// TIA Portal V17 export
// export: Created 2023-02-14T02:49:15.3088685Z, ExportSetting WithDefaults, DisplayName Totally Integrated Automation Portal, DisplayVersion V17, DisplayName TIA Portal Openness, DisplayVersion V17, DisplayName TIA Portal Teamcenter Gateway, DisplayVersion V17, DisplayName TIA Portal Version Control Interface, DisplayVersion V17, DisplayName SINAMICS Startdrive Advanced, DisplayVersion V17, DisplayName SINAMICS Startdrive G130, G150, S120, S150, SINAMICS MV, S210, DisplayVersion V17, DisplayName SINAMICS Startdrive G110M, G120, G120C, G120D, G120P, G115D, DisplayVersion V17, DisplayName STEP 7 Professional, DisplayVersion V17, DisplayName STEP 7 Safety, DisplayVersion V17, DisplayName WinCC Professional, DisplayVersion V17
DATA_BLOCK "CommSett_DB"   // DB10
{ S7_Optimized_Access := 'TRUE' }
VERSION : 0.1
// stored: AutoNumber false, DBAccessibleFromOPCUA true, DBAccessibleFromWebserver true, IsOnlyStoredInLoadMemory false, IsRetainMemResEnabled false, IsWriteProtectedInAS false, MemoryReserve 100
   VAR
      THE1_put : "typePut";
      THE1_get { S7_SetPoint := 'True'} : "typeGet";
      THE1_diagnostic { S7_SetPoint := 'True'} : "typeDiagnostic";
      THE2_put : "typePut";
      THE2_get { S7_SetPoint := 'True'} : "typeGet";
      THE2_diagnostic { S7_SetPoint := 'True'} : "typeDiagnostic";
      THE1_Comm_Error { S7_SetPoint := 'True'} : Bool;
      THE2_Comm_Error : Bool;
      THE1_Comm : Array[0..10] of Byte;
      THE2_Comm : Array[0..10] of Byte;
      CIP_put : "typePut";
      CIP_get { S7_SetPoint := 'True'} : "typeGet";
      CIP_diagnostic { S7_SetPoint := 'True'} : "typeDiagnostic";
      CIP_Comm_Error { S7_SetPoint := 'True'} : Bool;
      CIP_Comm : Array[0..10] of Byte;
   END_VAR
BEGIN
   THE1_put.connectionId := 16#100;
   THE1_get.connectionId := 16#100;
   THE2_put.connectionId := 16#101;
   THE2_get.connectionId := 16#101;
   CIP_put.connectionId := 16#102;
   CIP_get.connectionId := 16#102;
END_DATA_BLOCK
